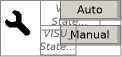
VISUALIZATION VISU_OperatingStatus  // 122x57
VAR_IN_OUT
	status : OperatingStatus;
	process : ChangeOperatingStateProcess;
END_VAR
    Frame (40,0 60x30)
        shows VISU_State_gray_green(state := status.auto)
    Button (60,0 60x20), "Auto", input disabled if: process.statuses.enabledStatus.disabled
        OnMouseClick: execute { process.set.state := OperatingStates.AUTO; process.do_request := TRUE; }
        OnMouseDown: execute {  }
    Button (60,25 60x20), "Manual", input disabled if: process.statuses.enabledStatus.disabled
        OnMouseClick: execute { process.set.state := OperatingStates.MANUAL; process.do_request := TRUE; }
        OnMouseDown: execute {  }
    Frame (40,25 36x30)
        shows VISU_State_gray_orange(state := status.manual)
    Polygon (9,27) (6,25) (5,22) (6,19) (11,22) (16,21) (16,16) (12,12) (14,10) (18,11) (21,14) (21,22) (29,30) (30,33) (28,35) (25,35) (17,27)
END_VISUALIZATION

(* stored: Version 1.1.0.1, ProductVersion 3.1.4019.2
   Visu VISU_OperatingStatus: Id {73d933c8-f1a9-4289-a205-6f6304bf9d40} *)
